FUNCTION_BLOCK L3_MachineManager (* Composite Function Block Type *)
  (* Standard: 61499-2 *)
  (* Version 0.0, 2014-10-06, EQUEROL, UJI *)
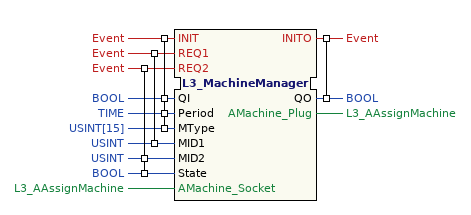
  EVENT_INPUT
    INIT WITH QI, MType, Period; (* Initialization Request *)
    REQ1 WITH MID1; (* Request to handle a released machine *)
    REQ2 WITH MID2, State; (* Request to handle a change in the operative state of a machine *)
  END_EVENT
  EVENT_OUTPUT
    INITO WITH QO; (* Initialization Confirm *)
  END_EVENT
  VAR_INPUT
    QI : BOOL; (* Input event qualifier *)
    Period : TIME := T#1000ms; (* MMCore execution period *)
    MType : ARRAY [0..14] OF USINT := [0,0,0,0,0,0,0,0,0,0,0,0,0,0,0]; (* Machine type vector *)
    MID1 : USINT; (* Machine identifier *)
    MID2 : USINT; (* Machine identifier *)
    State : BOOL; (* Machine state, true =OK, FALSE=KO *)
  END_VAR
  VAR_OUTPUT
    QO : BOOL; (* Output event qualifier *)
  END_VAR
  SOCKETS
    AMachine_Socket : L3_AAssignMachine;
  END_SOCKETS
  PLUGS
    AMachine_Plug : L3_AAssignMachine;
  END_PLUGS
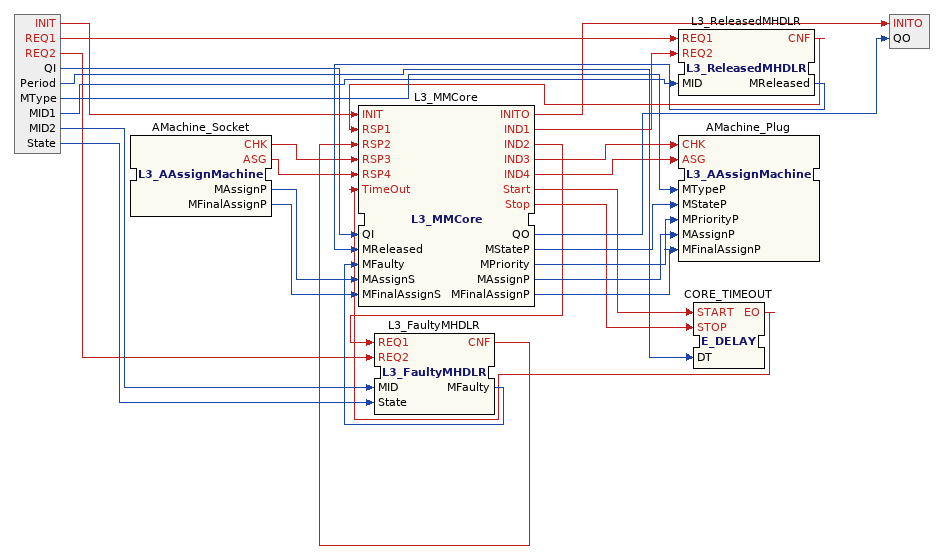
  FBS
    L3_ReleasedMHDLR : L3_ReleasedMHDLR;
    L3_FaultyMHDLR : L3_FaultyMHDLR;
    CORE_TIMEOUT : E_DELAY;
    L3_MMCore : L3_MMCore;
  END_FBS
  EVENT_CONNECTIONS
    REQ1 TO L3_ReleasedMHDLR.REQ1;
    REQ2 TO L3_FaultyMHDLR.REQ2;
    INIT TO L3_MMCore.INIT;
    L3_ReleasedMHDLR.CNF TO L3_MMCore.RSP1;
    L3_FaultyMHDLR.CNF TO L3_MMCore.RSP2;
    L3_MMCore.INITO TO INITO;
    L3_MMCore.IND1 TO L3_ReleasedMHDLR.REQ2;
    L3_MMCore.IND2 TO L3_FaultyMHDLR.REQ1;
    L3_MMCore.IND3 TO AMachine_Plug.CHK;
    L3_MMCore.IND4 TO AMachine_Plug.ASG;
    L3_MMCore.Start TO CORE_TIMEOUT.START;
    L3_MMCore.Stop TO CORE_TIMEOUT.STOP;
    CORE_TIMEOUT.EO TO L3_MMCore.TimeOut;
    AMachine_Socket.CHK TO L3_MMCore.RSP3;
    AMachine_Socket.ASG TO L3_MMCore.RSP4;
  END_CONNECTIONS
  DATA_CONNECTIONS
    MID1 TO L3_ReleasedMHDLR.MID;
    MID2 TO L3_FaultyMHDLR.MID;
    State TO L3_FaultyMHDLR.State;
    MType TO AMachine_Plug.MTypeP;
    QI TO L3_MMCore.QI;
    L3_ReleasedMHDLR.MReleased TO L3_MMCore.MReleased;
    L3_FaultyMHDLR.MFaulty TO L3_MMCore.MFaulty;
    L3_MMCore.QO TO QO;
    L3_MMCore.MStateP TO AMachine_Plug.MStateP;
    L3_MMCore.MPriority TO AMachine_Plug.MPriorityP;
    L3_MMCore.MAssignP TO AMachine_Plug.MAssignP;
    L3_MMCore.MFinalAssignP TO AMachine_Plug.MFinalAssignP;
    Period TO CORE_TIMEOUT.DT;
    AMachine_Socket.MAssignP TO L3_MMCore.MAssignS;
    AMachine_Socket.MFinalAssignP TO L3_MMCore.MFinalAssignS;
  END_CONNECTIONS
END_FUNCTION_BLOCK
